   // movePath.pathDataArray[4].commands[17].cmdParameters.pickAndPlaceParameters.targetParameter.direction[1..3] := 0.0;
   // movePath.pathDataArray[4].commands[18].cmdParameters.pickAndPlaceParameters.targetParameter.direction[1..3] := 0.0;
   // movePath.pathDataArray[4].commands[19].cmdParameters.pickAndPlaceParameters.targetParameter.direction[1..3] := 0.0;
   // movePath.pathDataArray[4].commands[20].cmdParameters.pickAndPlaceParameters.targetParameter.direction[1..3] := 0.0;
   // movePath.pathDataArray[5].commands[1].cmdParameters.pickAndPlaceParameters.targetParameter.direction[1..3] := 0.0;
   // movePath.pathDataArray[5].commands[2].cmdParameters.pickAndPlaceParameters.targetParameter.direction[1..3] := 0.0;
   // movePath.pathDataArray[5].commands[3].cmdParameters.pickAndPlaceParameters.targetParameter.direction[1..3] := 0.0;
   // movePath.pathDataArray[5].commands[4].cmdParameters.pickAndPlaceParameters.targetParameter.direction[1..3] := 0.0;
   // movePath.pathDataArray[5].commands[5].cmdParameters.pickAndPlaceParameters.targetParameter.direction[1..3] := 0.0;
   // movePath.pathDataArray[5].commands[6].cmdParameters.pickAndPlaceParameters.targetParameter.direction[1..3] := 0.0;
   // movePath.pathDataArray[5].commands[7].cmdParameters.pickAndPlaceParameters.targetParameter.direction[1..3] := 0.0;
   // movePath.pathDataArray[5].commands[8].cmdParameters.pickAndPlaceParameters.targetParameter.direction[1..3] := 0.0;
   // movePath.pathDataArray[5].commands[9].cmdParameters.pickAndPlaceParameters.targetParameter.direction[1..3] := 0.0;
   // movePath.pathDataArray[5].commands[10].cmdParameters.pickAndPlaceParameters.targetParameter.direction[1..3] := 0.0;
   // movePath.pathDataArray[5].commands[11].cmdParameters.pickAndPlaceParameters.targetParameter.direction[1..3] := 0.0;
   // movePath.pathDataArray[5].commands[12].cmdParameters.pickAndPlaceParameters.targetParameter.direction[1..3] := 0.0;
   // movePath.pathDataArray[5].commands[13].cmdParameters.pickAndPlaceParameters.targetParameter.direction[1..3] := 0.0;
   // movePath.pathDataArray[5].commands[14].cmdParameters.pickAndPlaceParameters.targetParameter.direction[1..3] := 0.0;
   // movePath.pathDataArray[5].commands[15].cmdParameters.pickAndPlaceParameters.targetParameter.direction[1..3] := 0.0;
   // movePath.pathDataArray[5].commands[16].cmdParameters.pickAndPlaceParameters.targetParameter.direction[1..3] := 0.0;
   // movePath.pathDataArray[5].commands[17].cmdParameters.pickAndPlaceParameters.targetParameter.direction[1..3] := 0.0;
   // movePath.pathDataArray[5].commands[18].cmdParameters.pickAndPlaceParameters.targetParameter.direction[1..3] := 0.0;
   // movePath.pathDataArray[5].commands[19].cmdParameters.pickAndPlaceParameters.targetParameter.direction[1..3] := 0.0;
   // movePath.pathDataArray[5].commands[20].cmdParameters.pickAndPlaceParameters.targetParameter.direction[1..3] := 0.0;
   // movePath.pathDataArray[1].commands[1..20].cmdParameters.pickAndPlaceParameters.targetParameter.workingHeight := 0.0;
   // movePath.pathDataArray[2].commands[1..20].cmdParameters.pickAndPlaceParameters.targetParameter.workingHeight := 0.0;
   // movePath.pathDataArray[3].commands[1..20].cmdParameters.pickAndPlaceParameters.targetParameter.workingHeight := 0.0;
   // movePath.pathDataArray[4].commands[1].cmdParameters.pickAndPlaceParameters.targetParameter.workingHeight := 0.0;
   // movePath.pathDataArray[4].commands[2].cmdParameters.pickAndPlaceParameters.targetParameter.workingHeight := 60.0;
   // movePath.pathDataArray[4].commands[3].cmdParameters.pickAndPlaceParameters.targetParameter.workingHeight := 0.0;
   // movePath.pathDataArray[4].commands[4].cmdParameters.pickAndPlaceParameters.targetParameter.workingHeight := 60.0;
   // movePath.pathDataArray[4].commands[5..20].cmdParameters.pickAndPlaceParameters.targetParameter.workingHeight := 0.0;
   // movePath.pathDataArray[5].commands[1..20].cmdParameters.pickAndPlaceParameters.targetParameter.workingHeight := 0.0;
   // movePath.pathDataArray[1].commands[1..20].cmdParameters.pickAndPlaceParameters.targetParameter.transitionArea := 0.0;
   // movePath.pathDataArray[2].commands[1..20].cmdParameters.pickAndPlaceParameters.targetParameter.transitionArea := 0.0;
   // movePath.pathDataArray[3].commands[1..20].cmdParameters.pickAndPlaceParameters.targetParameter.transitionArea := 0.0;
   // movePath.pathDataArray[4].commands[1..20].cmdParameters.pickAndPlaceParameters.targetParameter.transitionArea := 0.0;
   // movePath.pathDataArray[5].commands[1..20].cmdParameters.pickAndPlaceParameters.targetParameter.transitionArea := 0.0;
   // movePath.pathDataArray[1].commands[1..20].cmdParameters.pickAndPlaceParameters.targetParameter.dynamicsFactor := 100.0;
   // movePath.pathDataArray[2].commands[1..20].cmdParameters.pickAndPlaceParameters.targetParameter.dynamicsFactor := 100.0;
   // movePath.pathDataArray[3].commands[1..20].cmdParameters.pickAndPlaceParameters.targetParameter.dynamicsFactor := 100.0;
   // movePath.pathDataArray[4].commands[1..20].cmdParameters.pickAndPlaceParameters.targetParameter.dynamicsFactor := 100.0;
   // movePath.pathDataArray[5].commands[1..20].cmdParameters.pickAndPlaceParameters.targetParameter.dynamicsFactor := 100.0;
   // movePath.pathDataArray[1].commands[1].setFlags[1].flag := 1;
   // movePath.pathDataArray[1].commands[1].setFlags[2..3].flag := -1;
   // movePath.pathDataArray[1].commands[2].setFlags[1..3].flag := -1;
   // movePath.pathDataArray[1].commands[3].setFlags[1].flag := 0;
   // movePath.pathDataArray[1].commands[3].setFlags[2].flag := 1;
   // movePath.pathDataArray[1].commands[3].setFlags[3].flag := -1;
   // movePath.pathDataArray[1].commands[4].setFlags[1..3].flag := -1;
   // movePath.pathDataArray[1].commands[5].setFlags[1..3].flag := -1;
   // movePath.pathDataArray[1].commands[6].setFlags[1..3].flag := -1;
   // movePath.pathDataArray[1].commands[7].setFlags[1].flag := 0;
   // movePath.pathDataArray[1].commands[7].setFlags[2..3].flag := -1;
   // movePath.pathDataArray[1].commands[8].setFlags[1..3].flag := -1;
   // movePath.pathDataArray[1].commands[9].setFlags[1].flag := 1;
   // movePath.pathDataArray[1].commands[9].setFlags[2..3].flag := -1;
   // movePath.pathDataArray[1].commands[10].setFlags[1..3].flag := -1;
   // movePath.pathDataArray[1].commands[11].setFlags[1..3].flag := -1;
   // movePath.pathDataArray[1].commands[12].setFlags[1..3].flag := -1;
   // movePath.pathDataArray[1].commands[13].setFlags[1..3].flag := -1;
   // movePath.pathDataArray[1].commands[14].setFlags[1..3].flag := -1;
   // movePath.pathDataArray[1].commands[15].setFlags[1..3].flag := -1;
   // movePath.pathDataArray[1].commands[16].setFlags[1..3].flag := -1;
   // movePath.pathDataArray[1].commands[17].setFlags[1..3].flag := -1;
   // movePath.pathDataArray[1].commands[18].setFlags[1..3].flag := -1;
   // movePath.pathDataArray[1].commands[19].setFlags[1..3].flag := -1;
   // movePath.pathDataArray[1].commands[20].setFlags[1..3].flag := -1;
   // movePath.pathDataArray[2].commands[1].setFlags[1..3].flag := -1;
   // movePath.pathDataArray[2].commands[2].setFlags[1].flag := 1;
   // movePath.pathDataArray[2].commands[2].setFlags[2..3].flag := -1;
   // movePath.pathDataArray[2].commands[3].setFlags[1..3].flag := -1;
   // movePath.pathDataArray[2].commands[4].setFlags[1].flag := 0;
   // movePath.pathDataArray[2].commands[4].setFlags[2].flag := 1;
   // movePath.pathDataArray[2].commands[4].setFlags[3].flag := -1;
   // movePath.pathDataArray[2].commands[5].setFlags[1..3].flag := -1;
   // movePath.pathDataArray[2].commands[6].setFlags[1..3].flag := -1;
   // movePath.pathDataArray[2].commands[7].setFlags[1..3].flag := -1;
   // movePath.pathDataArray[2].commands[8].setFlags[1].flag := 0;
   // movePath.pathDataArray[2].commands[8].setFlags[2..3].flag := -1;
   // movePath.pathDataArray[2].commands[9].setFlags[1..3].flag := -1;
   // movePath.pathDataArray[2].commands[10].setFlags[1].flag := 1;
   // movePath.pathDataArray[2].commands[10].setFlags[2..3].flag := -1;
   // movePath.pathDataArray[2].commands[11].setFlags[1..3].flag := -1;
   // movePath.pathDataArray[2].commands[12].setFlags[1..3].flag := -1;
   // movePath.pathDataArray[2].commands[13].setFlags[1..3].flag := -1;
   // movePath.pathDataArray[2].commands[14].setFlags[1..3].flag := -1;
   // movePath.pathDataArray[2].commands[15].setFlags[1..3].flag := -1;
   // movePath.pathDataArray[2].commands[16].setFlags[1..3].flag := -1;
   // movePath.pathDataArray[2].commands[17].setFlags[1..3].flag := -1;
   // movePath.pathDataArray[2].commands[18].setFlags[1..3].flag := -1;
   // movePath.pathDataArray[2].commands[19].setFlags[1..3].flag := -1;
   // movePath.pathDataArray[2].commands[20].setFlags[1..3].flag := -1;
   // movePath.pathDataArray[3].commands[1].setFlags[1].flag := 2;
   // movePath.pathDataArray[3].commands[1].setFlags[2].flag := 3;
   // movePath.pathDataArray[3].commands[1].setFlags[3].flag := -1;
   // movePath.pathDataArray[3].commands[2].setFlags[1].flag := 4;
   // movePath.pathDataArray[3].commands[2].setFlags[2..3].flag := -1;
   // movePath.pathDataArray[3].commands[3].setFlags[1..3].flag := -1;
   // movePath.pathDataArray[3].commands[4].setFlags[1..3].flag := -1;
   // movePath.pathDataArray[3].commands[5].setFlags[1].flag := 3;
   // movePath.pathDataArray[3].commands[5].setFlags[2..3].flag := -1;
   // movePath.pathDataArray[3].commands[6].setFlags[1..3].flag := -1;
   // movePath.pathDataArray[3].commands[7].setFlags[1..3].flag := -1;
   // movePath.pathDataArray[3].commands[8].setFlags[1..3].flag := -1;
   // movePath.pathDataArray[3].commands[9].setFlags[1..3].flag := -1;
   // movePath.pathDataArray[3].commands[10].setFlags[1..3].flag := -1;
   // movePath.pathDataArray[3].commands[11].setFlags[1..3].flag := -1;
   // movePath.pathDataArray[3].commands[12].setFlags[1..3].flag := -1;
   // movePath.pathDataArray[3].commands[13].setFlags[1..3].flag := -1;
   // movePath.pathDataArray[3].commands[14].setFlags[1..3].flag := -1;
   // movePath.pathDataArray[3].commands[15].setFlags[1..3].flag := -1;
   // movePath.pathDataArray[3].commands[16].setFlags[1..3].flag := -1;
   // movePath.pathDataArray[3].commands[17].setFlags[1..3].flag := -1;
   // movePath.pathDataArray[3].commands[18].setFlags[1..3].flag := -1;
   // movePath.pathDataArray[3].commands[19].setFlags[1..3].flag := -1;
   // movePath.pathDataArray[3].commands[20].setFlags[1..3].flag := -1;
   // movePath.pathDataArray[4].commands[1].setFlags[1].flag := 5;
   // movePath.pathDataArray[4].commands[1].setFlags[2..3].flag := -1;
   // movePath.pathDataArray[4].commands[2].setFlags[1].flag := -1;
   // movePath.pathDataArray[4].commands[2].setFlags[2].flag := 5;
   // movePath.pathDataArray[4].commands[2].setFlags[3].flag := -1;
   // movePath.pathDataArray[4].commands[3].setFlags[1..3].flag := -1;
   // movePath.pathDataArray[4].commands[4].setFlags[1..3].flag := -1;
   // movePath.pathDataArray[4].commands[5].setFlags[1..3].flag := -1;
   // movePath.pathDataArray[4].commands[6].setFlags[1..3].flag := -1;
   // movePath.pathDataArray[4].commands[7].setFlags[1..3].flag := -1;
   // movePath.pathDataArray[4].commands[8].setFlags[1..3].flag := -1;
   // movePath.pathDataArray[4].commands[9].setFlags[1..3].flag := -1;
   // movePath.pathDataArray[4].commands[10].setFlags[1..3].flag := -1;
   // movePath.pathDataArray[4].commands[11].setFlags[1..3].flag := -1;
   // movePath.pathDataArray[4].commands[12].setFlags[1..3].flag := -1;
   // movePath.pathDataArray[4].commands[13].setFlags[1..3].flag := -1;
   // movePath.pathDataArray[4].commands[14].setFlags[1..3].flag := -1;
   // movePath.pathDataArray[4].commands[15].setFlags[1..3].flag := -1;
   // movePath.pathDataArray[4].commands[16].setFlags[1..3].flag := -1;
   // movePath.pathDataArray[4].commands[17].setFlags[1..3].flag := -1;
   // movePath.pathDataArray[4].commands[18].setFlags[1..3].flag := -1;
   // movePath.pathDataArray[4].commands[19].setFlags[1..3].flag := -1;
   // movePath.pathDataArray[4].commands[20].setFlags[1..3].flag := -1;
   // movePath.pathDataArray[5].commands[1].setFlags[1..3].flag := -1;
   // movePath.pathDataArray[5].commands[2].setFlags[1..3].flag := -1;
   // movePath.pathDataArray[5].commands[3].setFlags[1..3].flag := -1;
   // movePath.pathDataArray[5].commands[4].setFlags[1..3].flag := -1;
   // movePath.pathDataArray[5].commands[5].setFlags[1..3].flag := -1;
   // movePath.pathDataArray[5].commands[6].setFlags[1..3].flag := -1;
   // movePath.pathDataArray[5].commands[7].setFlags[1..3].flag := -1;
   // movePath.pathDataArray[5].commands[8].setFlags[1..3].flag := -1;
   // movePath.pathDataArray[5].commands[9].setFlags[1..3].flag := -1;
   // movePath.pathDataArray[5].commands[10].setFlags[1..3].flag := -1;
   // movePath.pathDataArray[5].commands[11].setFlags[1..3].flag := -1;
   // movePath.pathDataArray[5].commands[12].setFlags[1..3].flag := -1;
   // movePath.pathDataArray[5].commands[13].setFlags[1..3].flag := -1;
   // movePath.pathDataArray[5].commands[14].setFlags[1..3].flag := -1;
   // movePath.pathDataArray[5].commands[15].setFlags[1..3].flag := -1;
   // movePath.pathDataArray[5].commands[16].setFlags[1..3].flag := -1;
   // movePath.pathDataArray[5].commands[17].setFlags[1..3].flag := -1;
   // movePath.pathDataArray[5].commands[18].setFlags[1..3].flag := -1;
   // movePath.pathDataArray[5].commands[19].setFlags[1..3].flag := -1;
   // movePath.pathDataArray[5].commands[20].setFlags[1..3].flag := -1;
   // movePath.pathDataArray[1].commands[1].setFlags[1].flagMode := 1;
   // movePath.pathDataArray[1].commands[1].setFlags[2..3].flagMode := 0;
   // movePath.pathDataArray[1].commands[2].setFlags[1..3].flagMode := 1;
   // movePath.pathDataArray[1].commands[3].setFlags[1].flagMode := 1;
   // movePath.pathDataArray[1].commands[3].setFlags[2].flagMode := 11;
   // movePath.pathDataArray[1].commands[3].setFlags[3].flagMode := 1;
   // movePath.pathDataArray[1].commands[4].setFlags[1..3].flagMode := 1;
   // movePath.pathDataArray[1].commands[5].setFlags[1..3].flagMode := 1;
   // movePath.pathDataArray[1].commands[6].setFlags[1..3].flagMode := 1;
   // movePath.pathDataArray[1].commands[7].setFlags[1].flagMode := 1;
   // movePath.pathDataArray[1].commands[7].setFlags[2..3].flagMode := 0;
   // movePath.pathDataArray[1].commands[8].setFlags[1..3].flagMode := 0;
   // movePath.pathDataArray[1].commands[9].setFlags[1].flagMode := 11;
   // movePath.pathDataArray[1].commands[9].setFlags[2..3].flagMode := 0;
   // movePath.pathDataArray[1].commands[10].setFlags[1..3].flagMode := 1;
   // movePath.pathDataArray[1].commands[11].setFlags[1..3].flagMode := 1;
   // movePath.pathDataArray[1].commands[12].setFlags[1..3].flagMode := 1;
   // movePath.pathDataArray[1].commands[13].setFlags[1..3].flagMode := 1;
   // movePath.pathDataArray[1].commands[14].setFlags[1..3].flagMode := 1;
   // movePath.pathDataArray[1].commands[15].setFlags[1..3].flagMode := 1;
   // movePath.pathDataArray[1].commands[16].setFlags[1..3].flagMode := 1;
   // movePath.pathDataArray[1].commands[17].setFlags[1..3].flagMode := 1;
   // movePath.pathDataArray[1].commands[18].setFlags[1..3].flagMode := 1;
   // movePath.pathDataArray[1].commands[19].setFlags[1..3].flagMode := 1;
   // movePath.pathDataArray[1].commands[20].setFlags[1..3].flagMode := 1;
   // movePath.pathDataArray[2].commands[1].setFlags[1..3].flagMode := 1;
   // movePath.pathDataArray[2].commands[2].setFlags[1].flagMode := 1;
   // movePath.pathDataArray[2].commands[2].setFlags[2..3].flagMode := 0;
   // movePath.pathDataArray[2].commands[3].setFlags[1..3].flagMode := 1;
   // movePath.pathDataArray[2].commands[4].setFlags[1].flagMode := 1;
   // movePath.pathDataArray[2].commands[4].setFlags[2].flagMode := 11;
   // movePath.pathDataArray[2].commands[4].setFlags[3].flagMode := 1;
   // movePath.pathDataArray[2].commands[5].setFlags[1..3].flagMode := 1;
   // movePath.pathDataArray[2].commands[6].setFlags[1..3].flagMode := 1;
   // movePath.pathDataArray[2].commands[7].setFlags[1..3].flagMode := 1;
   // movePath.pathDataArray[2].commands[8].setFlags[1].flagMode := 1;
   // movePath.pathDataArray[2].commands[8].setFlags[2..3].flagMode := 0;
   // movePath.pathDataArray[2].commands[9].setFlags[1..3].flagMode := 0;
   // movePath.pathDataArray[2].commands[10].setFlags[1].flagMode := 11;
   // movePath.pathDataArray[2].commands[10].setFlags[2..3].flagMode := 0;
   // movePath.pathDataArray[2].commands[11].setFlags[1..3].flagMode := 1;
   // movePath.pathDataArray[2].commands[12].setFlags[1..3].flagMode := 1;
   // movePath.pathDataArray[2].commands[13].setFlags[1..3].flagMode := 1;
   // movePath.pathDataArray[2].commands[14].setFlags[1..3].flagMode := 1;
   // movePath.pathDataArray[2].commands[15].setFlags[1..3].flagMode := 1;
   // movePath.pathDataArray[2].commands[16].setFlags[1..3].flagMode := 1;
   // movePath.pathDataArray[2].commands[17].setFlags[1..3].flagMode := 1;
   // movePath.pathDataArray[2].commands[18].setFlags[1..3].flagMode := 1;
   // movePath.pathDataArray[2].commands[19].setFlags[1..3].flagMode := 1;
   // movePath.pathDataArray[2].commands[20].setFlags[1..3].flagMode := 1;
   // movePath.pathDataArray[3].commands[1].setFlags[1].flagMode := 26;
   // movePath.pathDataArray[3].commands[1].setFlags[2..3].flagMode := 1;
   // movePath.pathDataArray[3].commands[2].setFlags[1].flagMode := 11;
   // movePath.pathDataArray[3].commands[2].setFlags[2..3].flagMode := 1;
   // movePath.pathDataArray[3].commands[3].setFlags[1..3].flagMode := 1;
   // movePath.pathDataArray[3].commands[4].setFlags[1..3].flagMode := 1;
   // movePath.pathDataArray[3].commands[5].setFlags[1].flagMode := 11;
   // movePath.pathDataArray[3].commands[5].setFlags[2..3].flagMode := 1;
   // movePath.pathDataArray[3].commands[6].setFlags[1..3].flagMode := 1;
   // movePath.pathDataArray[3].commands[7].setFlags[1..3].flagMode := 1;
   // movePath.pathDataArray[3].commands[8].setFlags[1..3].flagMode := 1;
   // movePath.pathDataArray[3].commands[9].setFlags[1..3].flagMode := 1;
   // movePath.pathDataArray[3].commands[10].setFlags[1..3].flagMode := 1;
   // movePath.pathDataArray[3].commands[11].setFlags[1..3].flagMode := 1;
   // movePath.pathDataArray[3].commands[12].setFlags[1..3].flagMode := 1;
   // movePath.pathDataArray[3].commands[13].setFlags[1..3].flagMode := 1;
   // movePath.pathDataArray[3].commands[14].setFlags[1..3].flagMode := 1;
   // movePath.pathDataArray[3].commands[15].setFlags[1..3].flagMode := 1;
   // movePath.pathDataArray[3].commands[16].setFlags[1..3].flagMode := 1;
   // movePath.pathDataArray[3].commands[17].setFlags[1..3].flagMode := 1;
   // movePath.pathDataArray[3].commands[18].setFlags[1..3].flagMode := 1;
   // movePath.pathDataArray[3].commands[19].setFlags[1..3].flagMode := 1;
   // movePath.pathDataArray[3].commands[20].setFlags[1..3].flagMode := 1;
   // movePath.pathDataArray[4].commands[1].setFlags[1].flagMode := 26;
   // movePath.pathDataArray[4].commands[1].setFlags[2..3].flagMode := 1;
   // movePath.pathDataArray[4].commands[2].setFlags[1].flagMode := 1;
   // movePath.pathDataArray[4].commands[2].setFlags[2].flagMode := 21;
   // movePath.pathDataArray[4].commands[2].setFlags[3].flagMode := 1;
   // movePath.pathDataArray[4].commands[3].setFlags[1..3].flagMode := 1;
   // movePath.pathDataArray[4].commands[4].setFlags[1..3].flagMode := 1;
   // movePath.pathDataArray[4].commands[5].setFlags[1..3].flagMode := 1;
   // movePath.pathDataArray[4].commands[6].setFlags[1..3].flagMode := 1;
   // movePath.pathDataArray[4].commands[7].setFlags[1..3].flagMode := 1;
   // movePath.pathDataArray[4].commands[8].setFlags[1..3].flagMode := 1;
   // movePath.pathDataArray[4].commands[9].setFlags[1..3].flagMode := 1;
   // movePath.pathDataArray[4].commands[10].setFlags[1..3].flagMode := 1;
   // movePath.pathDataArray[4].commands[11].setFlags[1..3].flagMode := 1;
   // movePath.pathDataArray[4].commands[12].setFlags[1..3].flagMode := 1;
   // movePath.pathDataArray[4].commands[13].setFlags[1..3].flagMode := 1;
   // movePath.pathDataArray[4].commands[14].setFlags[1..3].flagMode := 1;
   // movePath.pathDataArray[4].commands[15].setFlags[1..3].flagMode := 1;
   // movePath.pathDataArray[4].commands[16].setFlags[1..3].flagMode := 1;
   // movePath.pathDataArray[4].commands[17].setFlags[1..3].flagMode := 1;
   // movePath.pathDataArray[4].commands[18].setFlags[1..3].flagMode := 1;
   // movePath.pathDataArray[4].commands[19].setFlags[1..3].flagMode := 1;
   // movePath.pathDataArray[4].commands[20].setFlags[1..3].flagMode := 1;
   // movePath.pathDataArray[5].commands[1].setFlags[1..3].flagMode := 1;
   // movePath.pathDataArray[5].commands[2].setFlags[1..3].flagMode := 1;
   // movePath.pathDataArray[5].commands[3].setFlags[1..3].flagMode := 1;
   // movePath.pathDataArray[5].commands[4].setFlags[1..3].flagMode := 1;
   // movePath.pathDataArray[5].commands[5].setFlags[1..3].flagMode := 1;
   // movePath.pathDataArray[5].commands[6].setFlags[1..3].flagMode := 1;
   // movePath.pathDataArray[5].commands[7].setFlags[1..3].flagMode := 1;
   // movePath.pathDataArray[5].commands[8].setFlags[1..3].flagMode := 1;
   // movePath.pathDataArray[5].commands[9].setFlags[1..3].flagMode := 1;
   // movePath.pathDataArray[5].commands[10].setFlags[1..3].flagMode := 1;
   // movePath.pathDataArray[5].commands[11].setFlags[1..3].flagMode := 1;
   // movePath.pathDataArray[5].commands[12].setFlags[1..3].flagMode := 1;
   // movePath.pathDataArray[5].commands[13].setFlags[1..3].flagMode := 1;
   // movePath.pathDataArray[5].commands[14].setFlags[1..3].flagMode := 1;
   // movePath.pathDataArray[5].commands[15].setFlags[1..3].flagMode := 1;
   // movePath.pathDataArray[5].commands[16].setFlags[1..3].flagMode := 1;
   // movePath.pathDataArray[5].commands[17].setFlags[1..3].flagMode := 1;
   // movePath.pathDataArray[5].commands[18].setFlags[1..3].flagMode := 1;
   // movePath.pathDataArray[5].commands[19].setFlags[1..3].flagMode := 1;
   // movePath.pathDataArray[5].commands[20].setFlags[1..3].flagMode := 1;
   // movePath.pathDataArray[1].commands[1].setFlags[1..3].remainingDistance := -1.0;
   // movePath.pathDataArray[1].commands[2].setFlags[1..3].remainingDistance := -1.0;
   // movePath.pathDataArray[1].commands[3].setFlags[1..3].remainingDistance := -1.0;
   // movePath.pathDataArray[1].commands[4].setFlags[1..3].remainingDistance := -1.0;
   // movePath.pathDataArray[1].commands[5].setFlags[1..3].remainingDistance := -1.0;
   // movePath.pathDataArray[1].commands[6].setFlags[1..3].remainingDistance := -1.0;
   // movePath.pathDataArray[1].commands[7].setFlags[1..3].remainingDistance := -1.0;
   // movePath.pathDataArray[1].commands[8].setFlags[1..3].remainingDistance := -1.0;
   // movePath.pathDataArray[1].commands[9].setFlags[1..3].remainingDistance := -1.0;
   // movePath.pathDataArray[1].commands[10].setFlags[1..3].remainingDistance := 0.0;
   // movePath.pathDataArray[1].commands[11].setFlags[1..3].remainingDistance := -1.0;
   // movePath.pathDataArray[1].commands[12].setFlags[1..3].remainingDistance := -1.0;
   // movePath.pathDataArray[1].commands[13].setFlags[1..3].remainingDistance := -1.0;
   // movePath.pathDataArray[1].commands[14].setFlags[1..3].remainingDistance := -1.0;
   // movePath.pathDataArray[1].commands[15].setFlags[1..3].remainingDistance := -1.0;
   // movePath.pathDataArray[1].commands[16].setFlags[1..3].remainingDistance := -1.0;
   // movePath.pathDataArray[1].commands[17].setFlags[1..3].remainingDistance := -1.0;
   // movePath.pathDataArray[1].commands[18].setFlags[1..3].remainingDistance := -1.0;
   // movePath.pathDataArray[1].commands[19].setFlags[1..3].remainingDistance := -1.0;
   // movePath.pathDataArray[1].commands[20].setFlags[1..3].remainingDistance := -1.0;
   // movePath.pathDataArray[2].commands[1].setFlags[1..3].remainingDistance := -1.0;
   // movePath.pathDataArray[2].commands[2].setFlags[1..3].remainingDistance := -1.0;
   // movePath.pathDataArray[2].commands[3].setFlags[1..3].remainingDistance := -1.0;
   // movePath.pathDataArray[2].commands[4].setFlags[1..3].remainingDistance := -1.0;
   // movePath.pathDataArray[2].commands[5].setFlags[1..3].remainingDistance := -1.0;
   // movePath.pathDataArray[2].commands[6].setFlags[1..3].remainingDistance := -1.0;
   // movePath.pathDataArray[2].commands[7].setFlags[1..3].remainingDistance := -1.0;
   // movePath.pathDataArray[2].commands[8].setFlags[1..3].remainingDistance := -1.0;
   // movePath.pathDataArray[2].commands[9].setFlags[1..3].remainingDistance := -1.0;
   // movePath.pathDataArray[2].commands[10].setFlags[1..3].remainingDistance := -1.0;
   // movePath.pathDataArray[2].commands[11].setFlags[1..3].remainingDistance := 0.0;
   // movePath.pathDataArray[2].commands[12].setFlags[1..3].remainingDistance := -1.0;
   // movePath.pathDataArray[2].commands[13].setFlags[1..3].remainingDistance := -1.0;
   // movePath.pathDataArray[2].commands[14].setFlags[1..3].remainingDistance := -1.0;
   // movePath.pathDataArray[2].commands[15].setFlags[1..3].remainingDistance := -1.0;
   // movePath.pathDataArray[2].commands[16].setFlags[1..3].remainingDistance := -1.0;
   // movePath.pathDataArray[2].commands[17].setFlags[1..3].remainingDistance := -1.0;
   // movePath.pathDataArray[2].commands[18].setFlags[1..3].remainingDistance := -1.0;
   // movePath.pathDataArray[2].commands[19].setFlags[1..3].remainingDistance := -1.0;
   // movePath.pathDataArray[2].commands[20].setFlags[1..3].remainingDistance := -1.0;
   // movePath.pathDataArray[3].commands[1].setFlags[1..3].remainingDistance := -1.0;
   // movePath.pathDataArray[3].commands[2].setFlags[1..3].remainingDistance := -1.0;
   // movePath.pathDataArray[3].commands[3].setFlags[1..3].remainingDistance := -1.0;
   // movePath.pathDataArray[3].commands[4].setFlags[1..3].remainingDistance := -1.0;
   // movePath.pathDataArray[3].commands[5].setFlags[1..3].remainingDistance := -1.0;
   // movePath.pathDataArray[3].commands[6].setFlags[1..3].remainingDistance := -1.0;
   // movePath.pathDataArray[3].commands[7].setFlags[1..3].remainingDistance := -1.0;
   // movePath.pathDataArray[3].commands[8].setFlags[1..3].remainingDistance := -1.0;
   // movePath.pathDataArray[3].commands[9].setFlags[1..3].remainingDistance := -1.0;
   // movePath.pathDataArray[3].commands[10].setFlags[1..3].remainingDistance := -1.0;
   // movePath.pathDataArray[3].commands[11].setFlags[1..3].remainingDistance := -1.0;
   // movePath.pathDataArray[3].commands[12].setFlags[1..3].remainingDistance := -1.0;
   // movePath.pathDataArray[3].commands[13].setFlags[1..3].remainingDistance := -1.0;
   // movePath.pathDataArray[3].commands[14].setFlags[1..3].remainingDistance := -1.0;
   // movePath.pathDataArray[3].commands[15].setFlags[1..3].remainingDistance := -1.0;
   // movePath.pathDataArray[3].commands[16].setFlags[1..3].remainingDistance := -1.0;
   // movePath.pathDataArray[3].commands[17].setFlags[1..3].remainingDistance := -1.0;
   // movePath.pathDataArray[3].commands[18].setFlags[1..3].remainingDistance := -1.0;
   // movePath.pathDataArray[3].commands[19].setFlags[1..3].remainingDistance := -1.0;
   // movePath.pathDataArray[3].commands[20].setFlags[1..3].remainingDistance := -1.0;
   // movePath.pathDataArray[4].commands[1].setFlags[1..3].remainingDistance := -1.0;
   // movePath.pathDataArray[4].commands[2].setFlags[1..3].remainingDistance := -1.0;
   // movePath.pathDataArray[4].commands[3].setFlags[1..3].remainingDistance := -1.0;
   // movePath.pathDataArray[4].commands[4].setFlags[1..3].remainingDistance := -1.0;
   // movePath.pathDataArray[4].commands[5].setFlags[1..3].remainingDistance := -1.0;
   // movePath.pathDataArray[4].commands[6].setFlags[1..3].remainingDistance := -1.0;
   // movePath.pathDataArray[4].commands[7].setFlags[1..3].remainingDistance := -1.0;
   // movePath.pathDataArray[4].commands[8].setFlags[1..3].remainingDistance := -1.0;
   // movePath.pathDataArray[4].commands[9].setFlags[1..3].remainingDistance := -1.0;
   // movePath.pathDataArray[4].commands[10].setFlags[1..3].remainingDistance := -1.0;
   // movePath.pathDataArray[4].commands[11].setFlags[1..3].remainingDistance := -1.0;
   // movePath.pathDataArray[4].commands[12].setFlags[1..3].remainingDistance := -1.0;
   // movePath.pathDataArray[4].commands[13].setFlags[1..3].remainingDistance := -1.0;
   // movePath.pathDataArray[4].commands[14].setFlags[1..3].remainingDistance := -1.0;
   // movePath.pathDataArray[4].commands[15].setFlags[1..3].remainingDistance := -1.0;
   // movePath.pathDataArray[4].commands[16].setFlags[1..3].remainingDistance := -1.0;
   // movePath.pathDataArray[4].commands[17].setFlags[1..3].remainingDistance := -1.0;
   // movePath.pathDataArray[4].commands[18].setFlags[1..3].remainingDistance := -1.0;
   // movePath.pathDataArray[4].commands[19].setFlags[1..3].remainingDistance := -1.0;
   // movePath.pathDataArray[4].commands[20].setFlags[1..3].remainingDistance := -1.0;
   // movePath.pathDataArray[5].commands[1].setFlags[1..3].remainingDistance := -1.0;
   // movePath.pathDataArray[5].commands[2].setFlags[1..3].remainingDistance := -1.0;
   // movePath.pathDataArray[5].commands[3].setFlags[1..3].remainingDistance := -1.0;
   // movePath.pathDataArray[5].commands[4].setFlags[1..3].remainingDistance := -1.0;
   // movePath.pathDataArray[5].commands[5].setFlags[1..3].remainingDistance := -1.0;
   // movePath.pathDataArray[5].commands[6].setFlags[1..3].remainingDistance := -1.0;
   // movePath.pathDataArray[5].commands[7].setFlags[1..3].remainingDistance := -1.0;
   // movePath.pathDataArray[5].commands[8].setFlags[1..3].remainingDistance := -1.0;
   // movePath.pathDataArray[5].commands[9].setFlags[1..3].remainingDistance := -1.0;
   // movePath.pathDataArray[5].commands[10].setFlags[1..3].remainingDistance := -1.0;
   // movePath.pathDataArray[5].commands[11].setFlags[1..3].remainingDistance := -1.0;
   // movePath.pathDataArray[5].commands[12].setFlags[1..3].remainingDistance := -1.0;
   // movePath.pathDataArray[5].commands[13].setFlags[1..3].remainingDistance := -1.0;
   // movePath.pathDataArray[5].commands[14].setFlags[1..3].remainingDistance := -1.0;
   // movePath.pathDataArray[5].commands[15].setFlags[1..3].remainingDistance := -1.0;
   // movePath.pathDataArray[5].commands[16].setFlags[1..3].remainingDistance := -1.0;
   // movePath.pathDataArray[5].commands[17].setFlags[1..3].remainingDistance := -1.0;
   // movePath.pathDataArray[5].commands[18].setFlags[1..3].remainingDistance := -1.0;
   // movePath.pathDataArray[5].commands[19].setFlags[1..3].remainingDistance := -1.0;
   // movePath.pathDataArray[5].commands[20].setFlags[1..3].remainingDistance := -1.0;
   // movePath.pathDataArray[1].commands[1].valueFlags[1..4].flag := -1;
   // movePath.pathDataArray[1].commands[2].valueFlags[1..4].flag := -1;
   // movePath.pathDataArray[1].commands[3].valueFlags[1..4].flag := -1;
   // movePath.pathDataArray[1].commands[4].valueFlags[1..4].flag := -1;
   // movePath.pathDataArray[1].commands[5].valueFlags[1..4].flag := -1;
   // movePath.pathDataArray[1].commands[6].valueFlags[1..4].flag := -1;
   // movePath.pathDataArray[1].commands[7].valueFlags[1..4].flag := -1;
   // movePath.pathDataArray[1].commands[8].valueFlags[1..4].flag := -1;
   // movePath.pathDataArray[1].commands[9].valueFlags[1..4].flag := -1;
   // movePath.pathDataArray[1].commands[10].valueFlags[1..4].flag := -1;
   // movePath.pathDataArray[1].commands[11].valueFlags[1..4].flag := -1;
   // movePath.pathDataArray[1].commands[12].valueFlags[1..4].flag := -1;
   // movePath.pathDataArray[1].commands[13].valueFlags[1..4].flag := -1;
   // movePath.pathDataArray[1].commands[14].valueFlags[1..4].flag := -1;
   // movePath.pathDataArray[1].commands[15].valueFlags[1..4].flag := -1;
   // movePath.pathDataArray[1].commands[16].valueFlags[1..4].flag := -1;
   // movePath.pathDataArray[1].commands[17].valueFlags[1..4].flag := -1;
   // movePath.pathDataArray[1].commands[18].valueFlags[1..4].flag := -1;
   // movePath.pathDataArray[1].commands[19].valueFlags[1..4].flag := -1;
   // movePath.pathDataArray[1].commands[20].valueFlags[1..4].flag := -1;
   // movePath.pathDataArray[2].commands[1].valueFlags[1..4].flag := -1;
   // movePath.pathDataArray[2].commands[2].valueFlags[1..4].flag := -1;
   // movePath.pathDataArray[2].commands[3].valueFlags[1..4].flag := -1;
   // movePath.pathDataArray[2].commands[4].valueFlags[1..4].flag := -1;
   // movePath.pathDataArray[2].commands[5].valueFlags[1..4].flag := -1;
   // movePath.pathDataArray[2].commands[6].valueFlags[1..4].flag := -1;
   // movePath.pathDataArray[2].commands[7].valueFlags[1..4].flag := -1;
   // movePath.pathDataArray[2].commands[8].valueFlags[1..4].flag := -1;
   // movePath.pathDataArray[2].commands[9].valueFlags[1..4].flag := -1;
   // movePath.pathDataArray[2].commands[10].valueFlags[1..4].flag := -1;
   // movePath.pathDataArray[2].commands[11].valueFlags[1..4].flag := -1;
   // movePath.pathDataArray[2].commands[12].valueFlags[1..4].flag := -1;
   // movePath.pathDataArray[2].commands[13].valueFlags[1..4].flag := -1;
   // movePath.pathDataArray[2].commands[14].valueFlags[1..4].flag := -1;
   // movePath.pathDataArray[2].commands[15].valueFlags[1..4].flag := -1;
   // movePath.pathDataArray[2].commands[16].valueFlags[1..4].flag := -1;
   // movePath.pathDataArray[2].commands[17].valueFlags[1..4].flag := -1;
   // movePath.pathDataArray[2].commands[18].valueFlags[1..4].flag := -1;
   // movePath.pathDataArray[2].commands[19].valueFlags[1..4].flag := -1;
   // movePath.pathDataArray[2].commands[20].valueFlags[1..4].flag := -1;
   // movePath.pathDataArray[3].commands[1].valueFlags[1..4].flag := -1;
   // movePath.pathDataArray[3].commands[2].valueFlags[1..4].flag := -1;
   // movePath.pathDataArray[3].commands[3].valueFlags[1..4].flag := -1;
   // movePath.pathDataArray[3].commands[4].valueFlags[1..4].flag := -1;
   // movePath.pathDataArray[3].commands[5].valueFlags[1..4].flag := -1;
   // movePath.pathDataArray[3].commands[6].valueFlags[1..4].flag := -1;
   // movePath.pathDataArray[3].commands[7].valueFlags[1..4].flag := -1;
   // movePath.pathDataArray[3].commands[8].valueFlags[1..4].flag := -1;
   // movePath.pathDataArray[3].commands[9].valueFlags[1..4].flag := -1;
   // movePath.pathDataArray[3].commands[10].valueFlags[1..4].flag := -1;
   // movePath.pathDataArray[3].commands[11].valueFlags[1..4].flag := -1;
   // movePath.pathDataArray[3].commands[12].valueFlags[1..4].flag := -1;
   // movePath.pathDataArray[3].commands[13].valueFlags[1..4].flag := -1;
   // movePath.pathDataArray[3].commands[14].valueFlags[1..4].flag := -1;
   // movePath.pathDataArray[3].commands[15].valueFlags[1..4].flag := -1;
   // movePath.pathDataArray[3].commands[16].valueFlags[1..4].flag := -1;
   // movePath.pathDataArray[3].commands[17].valueFlags[1..4].flag := -1;
   // movePath.pathDataArray[3].commands[18].valueFlags[1..4].flag := -1;
   // movePath.pathDataArray[3].commands[19].valueFlags[1..4].flag := -1;
   // movePath.pathDataArray[3].commands[20].valueFlags[1..4].flag := -1;
   // movePath.pathDataArray[4].commands[1].valueFlags[1..4].flag := -1;
   // movePath.pathDataArray[4].commands[2].valueFlags[1..4].flag := -1;
   // movePath.pathDataArray[4].commands[3].valueFlags[1..4].flag := -1;
   // movePath.pathDataArray[4].commands[4].valueFlags[1..4].flag := -1;
   // movePath.pathDataArray[4].commands[5].valueFlags[1..4].flag := -1;
   // movePath.pathDataArray[4].commands[6].valueFlags[1..4].flag := -1;
   // movePath.pathDataArray[4].commands[7].valueFlags[1..4].flag := -1;
   // movePath.pathDataArray[4].commands[8].valueFlags[1..4].flag := -1;
   // movePath.pathDataArray[4].commands[9].valueFlags[1..4].flag := -1;
   // movePath.pathDataArray[4].commands[10].valueFlags[1..4].flag := -1;
   // movePath.pathDataArray[4].commands[11].valueFlags[1..4].flag := -1;
   // movePath.pathDataArray[4].commands[12].valueFlags[1..4].flag := -1;
   // movePath.pathDataArray[4].commands[13].valueFlags[1..4].flag := -1;
   // movePath.pathDataArray[4].commands[14].valueFlags[1..4].flag := -1;
   // movePath.pathDataArray[4].commands[15].valueFlags[1..4].flag := -1;
   // movePath.pathDataArray[4].commands[16].valueFlags[1..4].flag := -1;
   // movePath.pathDataArray[4].commands[17].valueFlags[1..4].flag := -1;
   // movePath.pathDataArray[4].commands[18].valueFlags[1..4].flag := -1;
   // movePath.pathDataArray[4].commands[19].valueFlags[1..4].flag := -1;
   // movePath.pathDataArray[4].commands[20].valueFlags[1..4].flag := -1;
   // movePath.pathDataArray[5].commands[1].valueFlags[1..4].flag := -1;
   // movePath.pathDataArray[5].commands[2].valueFlags[1..4].flag := -1;
   // movePath.pathDataArray[5].commands[3].valueFlags[1..4].flag := -1;
   // movePath.pathDataArray[5].commands[4].valueFlags[1..4].flag := -1;
   // movePath.pathDataArray[5].commands[5].valueFlags[1..4].flag := -1;
   // movePath.pathDataArray[5].commands[6].valueFlags[1..4].flag := -1;
   // movePath.pathDataArray[5].commands[7].valueFlags[1..4].flag := -1;
   // movePath.pathDataArray[5].commands[8].valueFlags[1..4].flag := -1;
   // movePath.pathDataArray[5].commands[9].valueFlags[1..4].flag := -1;
   // movePath.pathDataArray[5].commands[10].valueFlags[1..4].flag := -1;
   // movePath.pathDataArray[5].commands[11].valueFlags[1..4].flag := -1;
   // movePath.pathDataArray[5].commands[12].valueFlags[1..4].flag := -1;
   // movePath.pathDataArray[5].commands[13].valueFlags[1..4].flag := -1;
   // movePath.pathDataArray[5].commands[14].valueFlags[1..4].flag := -1;
   // movePath.pathDataArray[5].commands[15].valueFlags[1..4].flag := -1;
   // movePath.pathDataArray[5].commands[16].valueFlags[1..4].flag := -1;
   // movePath.pathDataArray[5].commands[17].valueFlags[1..4].flag := -1;
   // movePath.pathDataArray[5].commands[18].valueFlags[1..4].flag := -1;
   // movePath.pathDataArray[5].commands[19].valueFlags[1..4].flag := -1;
   // movePath.pathDataArray[5].commands[20].valueFlags[1..4].flag := -1;
   // movePath.pathDataArray[1].commands[1].valueFlags[1..4].value := 0.0;
   // movePath.pathDataArray[1].commands[2].valueFlags[1..4].value := 0.0;
   // movePath.pathDataArray[1].commands[3].valueFlags[1..4].value := 0.0;
   // movePath.pathDataArray[1].commands[4].valueFlags[1..4].value := 0.0;
   // movePath.pathDataArray[1].commands[5].valueFlags[1..4].value := 0.0;
   // movePath.pathDataArray[1].commands[6].valueFlags[1..4].value := 0.0;
   // movePath.pathDataArray[1].commands[7].valueFlags[1..4].value := 0.0;
   // movePath.pathDataArray[1].commands[8].valueFlags[1..4].value := 0.0;
   // movePath.pathDataArray[1].commands[9].valueFlags[1..4].value := 0.0;
   // movePath.pathDataArray[1].commands[10].valueFlags[1..4].value := 0.0;
   // movePath.pathDataArray[1].commands[11].valueFlags[1..4].value := 0.0;
   // movePath.pathDataArray[1].commands[12].valueFlags[1..4].value := 0.0;
   // movePath.pathDataArray[1].commands[13].valueFlags[1..4].value := 0.0;
   // movePath.pathDataArray[1].commands[14].valueFlags[1..4].value := 0.0;
   // movePath.pathDataArray[1].commands[15].valueFlags[1..4].value := 0.0;
   // movePath.pathDataArray[1].commands[16].valueFlags[1..4].value := 0.0;
   // movePath.pathDataArray[1].commands[17].valueFlags[1..4].value := 0.0;
   // movePath.pathDataArray[1].commands[18].valueFlags[1..4].value := 0.0;
   // movePath.pathDataArray[1].commands[19].valueFlags[1..4].value := 0.0;
   // movePath.pathDataArray[1].commands[20].valueFlags[1..4].value := 0.0;
   // movePath.pathDataArray[2].commands[1].valueFlags[1..4].value := 0.0;
   // movePath.pathDataArray[2].commands[2].valueFlags[1..4].value := 0.0;
   // movePath.pathDataArray[2].commands[3].valueFlags[1..4].value := 0.0;
   // movePath.pathDataArray[2].commands[4].valueFlags[1..4].value := 0.0;
   // movePath.pathDataArray[2].commands[5].valueFlags[1..4].value := 0.0;
   // movePath.pathDataArray[2].commands[6].valueFlags[1..4].value := 0.0;
   // movePath.pathDataArray[2].commands[7].valueFlags[1..4].value := 0.0;
   // movePath.pathDataArray[2].commands[8].valueFlags[1..4].value := 0.0;
   // movePath.pathDataArray[2].commands[9].valueFlags[1..4].value := 0.0;
   // movePath.pathDataArray[2].commands[10].valueFlags[1..4].value := 0.0;
   // movePath.pathDataArray[2].commands[11].valueFlags[1..4].value := 0.0;
   // movePath.pathDataArray[2].commands[12].valueFlags[1..4].value := 0.0;
   // movePath.pathDataArray[2].commands[13].valueFlags[1..4].value := 0.0;
   // movePath.pathDataArray[2].commands[14].valueFlags[1..4].value := 0.0;
   // movePath.pathDataArray[2].commands[15].valueFlags[1..4].value := 0.0;
   // movePath.pathDataArray[2].commands[16].valueFlags[1..4].value := 0.0;
   // movePath.pathDataArray[2].commands[17].valueFlags[1..4].value := 0.0;
   // movePath.pathDataArray[2].commands[18].valueFlags[1..4].value := 0.0;
   // movePath.pathDataArray[2].commands[19].valueFlags[1..4].value := 0.0;
   // movePath.pathDataArray[2].commands[20].valueFlags[1..4].value := 0.0;
   // movePath.pathDataArray[3].commands[1].valueFlags[1..4].value := 0.0;
   // movePath.pathDataArray[3].commands[2].valueFlags[1..4].value := 0.0;
   // movePath.pathDataArray[3].commands[3].valueFlags[1..4].value := 0.0;
   // movePath.pathDataArray[3].commands[4].valueFlags[1..4].value := 0.0;
   // movePath.pathDataArray[3].commands[5].valueFlags[1..4].value := 0.0;
   // movePath.pathDataArray[3].commands[6].valueFlags[1..4].value := 0.0;
   // movePath.pathDataArray[3].commands[7].valueFlags[1..4].value := 0.0;
   // movePath.pathDataArray[3].commands[8].valueFlags[1..4].value := 0.0;
   // movePath.pathDataArray[3].commands[9].valueFlags[1..4].value := 0.0;
   // movePath.pathDataArray[3].commands[10].valueFlags[1..4].value := 0.0;
   // movePath.pathDataArray[3].commands[11].valueFlags[1..4].value := 0.0;
   // movePath.pathDataArray[3].commands[12].valueFlags[1..4].value := 0.0;
   // movePath.pathDataArray[3].commands[13].valueFlags[1..4].value := 0.0;
   // movePath.pathDataArray[3].commands[14].valueFlags[1..4].value := 0.0;
   // movePath.pathDataArray[3].commands[15].valueFlags[1..4].value := 0.0;
   // movePath.pathDataArray[3].commands[16].valueFlags[1..4].value := 0.0;
   // movePath.pathDataArray[3].commands[17].valueFlags[1..4].value := 0.0;
   // movePath.pathDataArray[3].commands[18].valueFlags[1..4].value := 0.0;
   // movePath.pathDataArray[3].commands[19].valueFlags[1..4].value := 0.0;
   // movePath.pathDataArray[3].commands[20].valueFlags[1..4].value := 0.0;
   // movePath.pathDataArray[4].commands[1].valueFlags[1..4].value := 0.0;
   // movePath.pathDataArray[4].commands[2].valueFlags[1..4].value := 0.0;
   // movePath.pathDataArray[4].commands[3].valueFlags[1..4].value := 0.0;
   // movePath.pathDataArray[4].commands[4].valueFlags[1..4].value := 0.0;
   // movePath.pathDataArray[4].commands[5].valueFlags[1..4].value := 0.0;
   // movePath.pathDataArray[4].commands[6].valueFlags[1..4].value := 0.0;
   // movePath.pathDataArray[4].commands[7].valueFlags[1..4].value := 0.0;
   // movePath.pathDataArray[4].commands[8].valueFlags[1..4].value := 0.0;
   // movePath.pathDataArray[4].commands[9].valueFlags[1..4].value := 0.0;
   // movePath.pathDataArray[4].commands[10].valueFlags[1..4].value := 0.0;
   // movePath.pathDataArray[4].commands[11].valueFlags[1..4].value := 0.0;
   // movePath.pathDataArray[4].commands[12].valueFlags[1..4].value := 0.0;
   // movePath.pathDataArray[4].commands[13].valueFlags[1..4].value := 0.0;
   // movePath.pathDataArray[4].commands[14].valueFlags[1..4].value := 0.0;
   // movePath.pathDataArray[4].commands[15].valueFlags[1..4].value := 0.0;
   // movePath.pathDataArray[4].commands[16].valueFlags[1..4].value := 0.0;
   // movePath.pathDataArray[4].commands[17].valueFlags[1..4].value := 0.0;
   // movePath.pathDataArray[4].commands[18].valueFlags[1..4].value := 0.0;
   // movePath.pathDataArray[4].commands[19].valueFlags[1..4].value := 0.0;
   // movePath.pathDataArray[4].commands[20].valueFlags[1..4].value := 0.0;
   // movePath.pathDataArray[5].commands[1].valueFlags[1..4].value := 0.0;
   // movePath.pathDataArray[5].commands[2].valueFlags[1..4].value := 0.0;
   // movePath.pathDataArray[5].commands[3].valueFlags[1..4].value := 0.0;
   // movePath.pathDataArray[5].commands[4].valueFlags[1..4].value := 0.0;
   // movePath.pathDataArray[5].commands[5].valueFlags[1..4].value := 0.0;
   // movePath.pathDataArray[5].commands[6].valueFlags[1..4].value := 0.0;
   // movePath.pathDataArray[5].commands[7].valueFlags[1..4].value := 0.0;
   // movePath.pathDataArray[5].commands[8].valueFlags[1..4].value := 0.0;
   // movePath.pathDataArray[5].commands[9].valueFlags[1..4].value := 0.0;
   // movePath.pathDataArray[5].commands[10].valueFlags[1..4].value := 0.0;
   // movePath.pathDataArray[5].commands[11].valueFlags[1..4].value := 0.0;
   // movePath.pathDataArray[5].commands[12].valueFlags[1..4].value := 0.0;
   // movePath.pathDataArray[5].commands[13].valueFlags[1..4].value := 0.0;
   // movePath.pathDataArray[5].commands[14].valueFlags[1..4].value := 0.0;
   // movePath.pathDataArray[5].commands[15].valueFlags[1..4].value := 0.0;
   // movePath.pathDataArray[5].commands[16].valueFlags[1..4].value := 0.0;
   // movePath.pathDataArray[5].commands[17].valueFlags[1..4].value := 0.0;
   // movePath.pathDataArray[5].commands[18].valueFlags[1..4].value := 0.0;
   // movePath.pathDataArray[5].commands[19].valueFlags[1..4].value := 0.0;
   // movePath.pathDataArray[5].commands[20].valueFlags[1..4].value := 0.0;
   // movePath.pathDataArray[1].commands[1].valueFlags[1..4].flagMode := 1;
   // movePath.pathDataArray[1].commands[2].valueFlags[1..4].flagMode := 1;
   // movePath.pathDataArray[1].commands[3].valueFlags[1..4].flagMode := 1;
   // movePath.pathDataArray[1].commands[4].valueFlags[1..4].flagMode := 1;
   // movePath.pathDataArray[1].commands[5].valueFlags[1..4].flagMode := 1;
   // movePath.pathDataArray[1].commands[6].valueFlags[1..4].flagMode := 1;
   // movePath.pathDataArray[1].commands[7].valueFlags[1..4].flagMode := 1;
   // movePath.pathDataArray[1].commands[8].valueFlags[1..4].flagMode := 1;
   // movePath.pathDataArray[1].commands[9].valueFlags[1..4].flagMode := 1;
   // movePath.pathDataArray[1].commands[10].valueFlags[1..4].flagMode := 1;
   // movePath.pathDataArray[1].commands[11].valueFlags[1..4].flagMode := 1;
   // movePath.pathDataArray[1].commands[12].valueFlags[1..4].flagMode := 1;
   // movePath.pathDataArray[1].commands[13].valueFlags[1..4].flagMode := 1;
   // movePath.pathDataArray[1].commands[14].valueFlags[1..4].flagMode := 1;
   // movePath.pathDataArray[1].commands[15].valueFlags[1..4].flagMode := 1;
   // movePath.pathDataArray[1].commands[16].valueFlags[1..4].flagMode := 1;
   // movePath.pathDataArray[1].commands[17].valueFlags[1..4].flagMode := 1;
   // movePath.pathDataArray[1].commands[18].valueFlags[1..4].flagMode := 1;
   // movePath.pathDataArray[1].commands[19].valueFlags[1..4].flagMode := 1;
   // movePath.pathDataArray[1].commands[20].valueFlags[1..4].flagMode := 1;
   // movePath.pathDataArray[2].commands[1].valueFlags[1..4].flagMode := 1;
   // movePath.pathDataArray[2].commands[2].valueFlags[1..4].flagMode := 1;
   // movePath.pathDataArray[2].commands[3].valueFlags[1..4].flagMode := 1;
   // movePath.pathDataArray[2].commands[4].valueFlags[1..4].flagMode := 1;
   // movePath.pathDataArray[2].commands[5].valueFlags[1..4].flagMode := 1;
   // movePath.pathDataArray[2].commands[6].valueFlags[1..4].flagMode := 1;
   // movePath.pathDataArray[2].commands[7].valueFlags[1..4].flagMode := 1;
   // movePath.pathDataArray[2].commands[8].valueFlags[1..4].flagMode := 1;
   // movePath.pathDataArray[2].commands[9].valueFlags[1..4].flagMode := 1;
   // movePath.pathDataArray[2].commands[10].valueFlags[1..4].flagMode := 1;
   // movePath.pathDataArray[2].commands[11].valueFlags[1..4].flagMode := 1;
   // movePath.pathDataArray[2].commands[12].valueFlags[1..4].flagMode := 1;
   // movePath.pathDataArray[2].commands[13].valueFlags[1..4].flagMode := 1;
   // movePath.pathDataArray[2].commands[14].valueFlags[1..4].flagMode := 1;
   // movePath.pathDataArray[2].commands[15].valueFlags[1..4].flagMode := 1;
   // movePath.pathDataArray[2].commands[16].valueFlags[1..4].flagMode := 1;
   // movePath.pathDataArray[2].commands[17].valueFlags[1..4].flagMode := 1;
   // movePath.pathDataArray[2].commands[18].valueFlags[1..4].flagMode := 1;
   // movePath.pathDataArray[2].commands[19].valueFlags[1..4].flagMode := 1;
   // movePath.pathDataArray[2].commands[20].valueFlags[1..4].flagMode := 1;
   // movePath.pathDataArray[3].commands[1].valueFlags[1..4].flagMode := 1;
   // movePath.pathDataArray[3].commands[2].valueFlags[1..4].flagMode := 1;
   // movePath.pathDataArray[3].commands[3].valueFlags[1..4].flagMode := 1;
   // movePath.pathDataArray[3].commands[4].valueFlags[1..4].flagMode := 1;
   // movePath.pathDataArray[3].commands[5].valueFlags[1..4].flagMode := 1;
   // movePath.pathDataArray[3].commands[6].valueFlags[1..4].flagMode := 1;
   // movePath.pathDataArray[3].commands[7].valueFlags[1..4].flagMode := 1;
   // movePath.pathDataArray[3].commands[8].valueFlags[1..4].flagMode := 1;
   // movePath.pathDataArray[3].commands[9].valueFlags[1..4].flagMode := 1;
   // movePath.pathDataArray[3].commands[10].valueFlags[1..4].flagMode := 1;
   // movePath.pathDataArray[3].commands[11].valueFlags[1..4].flagMode := 1;
   // movePath.pathDataArray[3].commands[12].valueFlags[1..4].flagMode := 1;
   // movePath.pathDataArray[3].commands[13].valueFlags[1..4].flagMode := 1;
   // movePath.pathDataArray[3].commands[14].valueFlags[1..4].flagMode := 1;
   // movePath.pathDataArray[3].commands[15].valueFlags[1..4].flagMode := 1;
   // movePath.pathDataArray[3].commands[16].valueFlags[1..4].flagMode := 1;
   // movePath.pathDataArray[3].commands[17].valueFlags[1..4].flagMode := 1;
   // movePath.pathDataArray[3].commands[18].valueFlags[1..4].flagMode := 1;
   // movePath.pathDataArray[3].commands[19].valueFlags[1..4].flagMode := 1;
   // movePath.pathDataArray[3].commands[20].valueFlags[1..4].flagMode := 1;
   // movePath.pathDataArray[4].commands[1].valueFlags[1..4].flagMode := 1;
   // movePath.pathDataArray[4].commands[2].valueFlags[1..4].flagMode := 1;
   // movePath.pathDataArray[4].commands[3].valueFlags[1..4].flagMode := 1;
   // movePath.pathDataArray[4].commands[4].valueFlags[1..4].flagMode := 1;
   // movePath.pathDataArray[4].commands[5].valueFlags[1..4].flagMode := 1;
   // movePath.pathDataArray[4].commands[6].valueFlags[1..4].flagMode := 1;
   // movePath.pathDataArray[4].commands[7].valueFlags[1..4].flagMode := 1;
   // movePath.pathDataArray[4].commands[8].valueFlags[1..4].flagMode := 1;
   // movePath.pathDataArray[4].commands[9].valueFlags[1..4].flagMode := 1;
   // movePath.pathDataArray[4].commands[10].valueFlags[1..4].flagMode := 1;
   // movePath.pathDataArray[4].commands[11].valueFlags[1..4].flagMode := 1;
   // movePath.pathDataArray[4].commands[12].valueFlags[1..4].flagMode := 1;
   // movePath.pathDataArray[4].commands[13].valueFlags[1..4].flagMode := 1;
   // movePath.pathDataArray[4].commands[14].valueFlags[1..4].flagMode := 1;
   // movePath.pathDataArray[4].commands[15].valueFlags[1..4].flagMode := 1;
   // movePath.pathDataArray[4].commands[16].valueFlags[1..4].flagMode := 1;
   // movePath.pathDataArray[4].commands[17].valueFlags[1..4].flagMode := 1;
   // movePath.pathDataArray[4].commands[18].valueFlags[1..4].flagMode := 1;
   // movePath.pathDataArray[4].commands[19].valueFlags[1..4].flagMode := 1;
   // movePath.pathDataArray[4].commands[20].valueFlags[1..4].flagMode := 1;
   // movePath.pathDataArray[5].commands[1].valueFlags[1..4].flagMode := 1;
   // movePath.pathDataArray[5].commands[2].valueFlags[1..4].flagMode := 1;
   // movePath.pathDataArray[5].commands[3].valueFlags[1..4].flagMode := 1;
   // movePath.pathDataArray[5].commands[4].valueFlags[1..4].flagMode := 1;
   // movePath.pathDataArray[5].commands[5].valueFlags[1..4].flagMode := 1;
   // movePath.pathDataArray[5].commands[6].valueFlags[1..4].flagMode := 1;
   // movePath.pathDataArray[5].commands[7].valueFlags[1..4].flagMode := 1;
   // movePath.pathDataArray[5].commands[8].valueFlags[1..4].flagMode := 1;
   // movePath.pathDataArray[5].commands[9].valueFlags[1..4].flagMode := 1;
   // movePath.pathDataArray[5].commands[10].valueFlags[1..4].flagMode := 1;
   // movePath.pathDataArray[5].commands[11].valueFlags[1..4].flagMode := 1;
   // movePath.pathDataArray[5].commands[12].valueFlags[1..4].flagMode := 1;
   // movePath.pathDataArray[5].commands[13].valueFlags[1..4].flagMode := 1;
   // movePath.pathDataArray[5].commands[14].valueFlags[1..4].flagMode := 1;
   // movePath.pathDataArray[5].commands[15].valueFlags[1..4].flagMode := 1;
   // movePath.pathDataArray[5].commands[16].valueFlags[1..4].flagMode := 1;
   // movePath.pathDataArray[5].commands[17].valueFlags[1..4].flagMode := 1;
   // movePath.pathDataArray[5].commands[18].valueFlags[1..4].flagMode := 1;
   // movePath.pathDataArray[5].commands[19].valueFlags[1..4].flagMode := 1;
   // movePath.pathDataArray[5].commands[20].valueFlags[1..4].flagMode := 1;
   // movePath.pathDataArray[1].commands[1].valueFlags[1..4].remainingDistance := -1.0;
   // movePath.pathDataArray[1].commands[2].valueFlags[1..4].remainingDistance := -1.0;
   // movePath.pathDataArray[1].commands[3].valueFlags[1..4].remainingDistance := -1.0;
   // movePath.pathDataArray[1].commands[4].valueFlags[1..4].remainingDistance := -1.0;
   // movePath.pathDataArray[1].commands[5].valueFlags[1..4].remainingDistance := -1.0;
   // movePath.pathDataArray[1].commands[6].valueFlags[1..4].remainingDistance := -1.0;
   // movePath.pathDataArray[1].commands[7].valueFlags[1..4].remainingDistance := -1.0;
   // movePath.pathDataArray[1].commands[8].valueFlags[1..4].remainingDistance := -1.0;
   // movePath.pathDataArray[1].commands[9].valueFlags[1..4].remainingDistance := -1.0;
   // movePath.pathDataArray[1].commands[10].valueFlags[1..4].remainingDistance := 0.0;
   // movePath.pathDataArray[1].commands[11].valueFlags[1..4].remainingDistance := -1.0;
   // movePath.pathDataArray[1].commands[12].valueFlags[1..4].remainingDistance := -1.0;
   // movePath.pathDataArray[1].commands[13].valueFlags[1..4].remainingDistance := -1.0;
   // movePath.pathDataArray[1].commands[14].valueFlags[1..4].remainingDistance := -1.0;
   // movePath.pathDataArray[1].commands[15].valueFlags[1..4].remainingDistance := -1.0;
   // movePath.pathDataArray[1].commands[16].valueFlags[1..4].remainingDistance := -1.0;
   // movePath.pathDataArray[1].commands[17].valueFlags[1..4].remainingDistance := -1.0;
   // movePath.pathDataArray[1].commands[18].valueFlags[1..4].remainingDistance := -1.0;
   // movePath.pathDataArray[1].commands[19].valueFlags[1..4].remainingDistance := -1.0;
   // movePath.pathDataArray[1].commands[20].valueFlags[1..4].remainingDistance := -1.0;
   // movePath.pathDataArray[2].commands[1].valueFlags[1..4].remainingDistance := -1.0;
   // movePath.pathDataArray[2].commands[2].valueFlags[1..4].remainingDistance := -1.0;
   // movePath.pathDataArray[2].commands[3].valueFlags[1..4].remainingDistance := -1.0;
   // movePath.pathDataArray[2].commands[4].valueFlags[1..4].remainingDistance := -1.0;
   // movePath.pathDataArray[2].commands[5].valueFlags[1..4].remainingDistance := -1.0;
   // movePath.pathDataArray[2].commands[6].valueFlags[1..4].remainingDistance := -1.0;
   // movePath.pathDataArray[2].commands[7].valueFlags[1..4].remainingDistance := -1.0;
   // movePath.pathDataArray[2].commands[8].valueFlags[1..4].remainingDistance := -1.0;
   // movePath.pathDataArray[2].commands[9].valueFlags[1..4].remainingDistance := -1.0;
   // movePath.pathDataArray[2].commands[10].valueFlags[1..4].remainingDistance := -1.0;
   // movePath.pathDataArray[2].commands[11].valueFlags[1..4].remainingDistance := 0.0;
   // movePath.pathDataArray[2].commands[12].valueFlags[1..4].remainingDistance := -1.0;
   // movePath.pathDataArray[2].commands[13].valueFlags[1..4].remainingDistance := -1.0;
   // movePath.pathDataArray[2].commands[14].valueFlags[1..4].remainingDistance := -1.0;
   // movePath.pathDataArray[2].commands[15].valueFlags[1..4].remainingDistance := -1.0;
   // movePath.pathDataArray[2].commands[16].valueFlags[1..4].remainingDistance := -1.0;
   // movePath.pathDataArray[2].commands[17].valueFlags[1..4].remainingDistance := -1.0;
   // movePath.pathDataArray[2].commands[18].valueFlags[1..4].remainingDistance := -1.0;
   // movePath.pathDataArray[2].commands[19].valueFlags[1..4].remainingDistance := -1.0;
   // movePath.pathDataArray[2].commands[20].valueFlags[1..4].remainingDistance := -1.0;
   // movePath.pathDataArray[3].commands[1].valueFlags[1..4].remainingDistance := -1.0;
   // movePath.pathDataArray[3].commands[2].valueFlags[1..4].remainingDistance := -1.0;
   // movePath.pathDataArray[3].commands[3].valueFlags[1..4].remainingDistance := -1.0;
   // movePath.pathDataArray[3].commands[4].valueFlags[1..4].remainingDistance := -1.0;
   // movePath.pathDataArray[3].commands[5].valueFlags[1..4].remainingDistance := -1.0;
   // movePath.pathDataArray[3].commands[6].valueFlags[1..4].remainingDistance := -1.0;
   // movePath.pathDataArray[3].commands[7].valueFlags[1..4].remainingDistance := -1.0;
   // movePath.pathDataArray[3].commands[8].valueFlags[1..4].remainingDistance := -1.0;
   // movePath.pathDataArray[3].commands[9].valueFlags[1..4].remainingDistance := -1.0;
   // movePath.pathDataArray[3].commands[10].valueFlags[1..4].remainingDistance := -1.0;
   // movePath.pathDataArray[3].commands[11].valueFlags[1..4].remainingDistance := -1.0;
   // movePath.pathDataArray[3].commands[12].valueFlags[1..4].remainingDistance := -1.0;
   // movePath.pathDataArray[3].commands[13].valueFlags[1..4].remainingDistance := -1.0;
   // movePath.pathDataArray[3].commands[14].valueFlags[1..4].remainingDistance := -1.0;
   // movePath.pathDataArray[3].commands[15].valueFlags[1..4].remainingDistance := -1.0;
   // movePath.pathDataArray[3].commands[16].valueFlags[1..4].remainingDistance := -1.0;
   // movePath.pathDataArray[3].commands[17].valueFlags[1..4].remainingDistance := -1.0;
   // movePath.pathDataArray[3].commands[18].valueFlags[1..4].remainingDistance := -1.0;
   // movePath.pathDataArray[3].commands[19].valueFlags[1..4].remainingDistance := -1.0;
   // movePath.pathDataArray[3].commands[20].valueFlags[1..4].remainingDistance := -1.0;
   // movePath.pathDataArray[4].commands[1].valueFlags[1..4].remainingDistance := -1.0;
   // movePath.pathDataArray[4].commands[2].valueFlags[1..4].remainingDistance := -1.0;
   // movePath.pathDataArray[4].commands[3].valueFlags[1..4].remainingDistance := -1.0;
   // movePath.pathDataArray[4].commands[4].valueFlags[1..4].remainingDistance := -1.0;
   // movePath.pathDataArray[4].commands[5].valueFlags[1..4].remainingDistance := -1.0;
   // movePath.pathDataArray[4].commands[6].valueFlags[1..4].remainingDistance := -1.0;
   // movePath.pathDataArray[4].commands[7].valueFlags[1..4].remainingDistance := -1.0;
   // movePath.pathDataArray[4].commands[8].valueFlags[1..4].remainingDistance := -1.0;
   // movePath.pathDataArray[4].commands[9].valueFlags[1..4].remainingDistance := -1.0;
   // movePath.pathDataArray[4].commands[10].valueFlags[1..4].remainingDistance := -1.0;
   // movePath.pathDataArray[4].commands[11].valueFlags[1..4].remainingDistance := -1.0;
   // movePath.pathDataArray[4].commands[12].valueFlags[1..4].remainingDistance := -1.0;
   // movePath.pathDataArray[4].commands[13].valueFlags[1..4].remainingDistance := -1.0;
   // movePath.pathDataArray[4].commands[14].valueFlags[1..4].remainingDistance := -1.0;
   // movePath.pathDataArray[4].commands[15].valueFlags[1..4].remainingDistance := -1.0;
   // movePath.pathDataArray[4].commands[16].valueFlags[1..4].remainingDistance := -1.0;
   // movePath.pathDataArray[4].commands[17].valueFlags[1..4].remainingDistance := -1.0;
   // movePath.pathDataArray[4].commands[18].valueFlags[1..4].remainingDistance := -1.0;
   // movePath.pathDataArray[4].commands[19].valueFlags[1..4].remainingDistance := -1.0;
   // movePath.pathDataArray[4].commands[20].valueFlags[1..4].remainingDistance := -1.0;
   // movePath.pathDataArray[5].commands[1].valueFlags[1..4].remainingDistance := -1.0;
   // movePath.pathDataArray[5].commands[2].valueFlags[1..4].remainingDistance := -1.0;
   // movePath.pathDataArray[5].commands[3].valueFlags[1..4].remainingDistance := -1.0;
   // movePath.pathDataArray[5].commands[4].valueFlags[1..4].remainingDistance := -1.0;
   // movePath.pathDataArray[5].commands[5].valueFlags[1..4].remainingDistance := -1.0;
   // movePath.pathDataArray[5].commands[6].valueFlags[1..4].remainingDistance := -1.0;
   // movePath.pathDataArray[5].commands[7].valueFlags[1..4].remainingDistance := -1.0;
   // movePath.pathDataArray[5].commands[8].valueFlags[1..4].remainingDistance := -1.0;
   // movePath.pathDataArray[5].commands[9].valueFlags[1..4].remainingDistance := -1.0;
   // movePath.pathDataArray[5].commands[10].valueFlags[1..4].remainingDistance := -1.0;
   // movePath.pathDataArray[5].commands[11].valueFlags[1..4].remainingDistance := -1.0;
   // movePath.pathDataArray[5].commands[12].valueFlags[1..4].remainingDistance := -1.0;
   // movePath.pathDataArray[5].commands[13].valueFlags[1..4].remainingDistance := -1.0;
   // movePath.pathDataArray[5].commands[14].valueFlags[1..4].remainingDistance := -1.0;
   // movePath.pathDataArray[5].commands[15].valueFlags[1..4].remainingDistance := -1.0;
   // movePath.pathDataArray[5].commands[16].valueFlags[1..4].remainingDistance := -1.0;
   // movePath.pathDataArray[5].commands[17].valueFlags[1..4].remainingDistance := -1.0;
   // movePath.pathDataArray[5].commands[18].valueFlags[1..4].remainingDistance := -1.0;
   // movePath.pathDataArray[5].commands[19].valueFlags[1..4].remainingDistance := -1.0;
   // movePath.pathDataArray[5].commands[20].valueFlags[1..4].remainingDistance := -1.0;
   // movePath.pathDataArray[1].commands[1].parameterValid[1..6] := TRUE;
   // movePath.pathDataArray[1].commands[2].parameterValid[1..6] := TRUE;
   // movePath.pathDataArray[1].commands[3].parameterValid[1..6] := TRUE;
   // movePath.pathDataArray[1].commands[4].parameterValid[1..6] := TRUE;
   // movePath.pathDataArray[1].commands[5].parameterValid[1..6] := TRUE;
   // movePath.pathDataArray[1].commands[6].parameterValid[1..6] := TRUE;
   // movePath.pathDataArray[1].commands[7].parameterValid[1..6] := TRUE;
   // movePath.pathDataArray[1].commands[8].parameterValid[1..6] := TRUE;
   // movePath.pathDataArray[1].commands[9].parameterValid[1..6] := TRUE;
   // movePath.pathDataArray[1].commands[10].parameterValid[1..6] := TRUE;
   // movePath.pathDataArray[1].commands[11].parameterValid[1..6] := TRUE;
   // movePath.pathDataArray[1].commands[12].parameterValid[1..6] := TRUE;
   // movePath.pathDataArray[1].commands[13].parameterValid[1..6] := TRUE;
   // movePath.pathDataArray[1].commands[14].parameterValid[1..6] := TRUE;
   // movePath.pathDataArray[1].commands[15].parameterValid[1..6] := TRUE;
   // movePath.pathDataArray[1].commands[16].parameterValid[1..6] := TRUE;
   // movePath.pathDataArray[1].commands[17].parameterValid[1..6] := TRUE;
   // movePath.pathDataArray[1].commands[18].parameterValid[1..6] := TRUE;
   // movePath.pathDataArray[1].commands[19].parameterValid[1..6] := TRUE;
   // movePath.pathDataArray[1].commands[20].parameterValid[1..6] := TRUE;
   // movePath.pathDataArray[2].commands[1].parameterValid[1..6] := TRUE;
   // movePath.pathDataArray[2].commands[2].parameterValid[1..6] := TRUE;
   // movePath.pathDataArray[2].commands[3].parameterValid[1..6] := TRUE;
   // movePath.pathDataArray[2].commands[4].parameterValid[1..6] := TRUE;
   // movePath.pathDataArray[2].commands[5].parameterValid[1..6] := TRUE;
   // movePath.pathDataArray[2].commands[6].parameterValid[1..6] := TRUE;
   // movePath.pathDataArray[2].commands[7].parameterValid[1..6] := TRUE;
   // movePath.pathDataArray[2].commands[8].parameterValid[1..6] := TRUE;
   // movePath.pathDataArray[2].commands[9].parameterValid[1..6] := TRUE;
   // movePath.pathDataArray[2].commands[10].parameterValid[1..6] := TRUE;
   // movePath.pathDataArray[2].commands[11].parameterValid[1..6] := TRUE;
   // movePath.pathDataArray[2].commands[12].parameterValid[1..6] := TRUE;
   // movePath.pathDataArray[2].commands[13].parameterValid[1..6] := TRUE;
   // movePath.pathDataArray[2].commands[14].parameterValid[1..6] := TRUE;
   // movePath.pathDataArray[2].commands[15].parameterValid[1..6] := TRUE;
   // movePath.pathDataArray[2].commands[16].parameterValid[1..6] := TRUE;
   // movePath.pathDataArray[2].commands[17].parameterValid[1..6] := TRUE;
   // movePath.pathDataArray[2].commands[18].parameterValid[1..6] := TRUE;
   // movePath.pathDataArray[2].commands[19].parameterValid[1..6] := TRUE;
   // movePath.pathDataArray[2].commands[20].parameterValid[1..6] := TRUE;
   // movePath.pathDataArray[3].commands[1].parameterValid[1..6] := TRUE;
   // movePath.pathDataArray[3].commands[2].parameterValid[1..6] := TRUE;
   // movePath.pathDataArray[3].commands[3].parameterValid[1..6] := TRUE;
   // movePath.pathDataArray[3].commands[4].parameterValid[1..6] := TRUE;
   // movePath.pathDataArray[3].commands[5].parameterValid[1..6] := TRUE;
   // movePath.pathDataArray[3].commands[6].parameterValid[1..6] := TRUE;
   // movePath.pathDataArray[3].commands[7].parameterValid[1..6] := TRUE;
   // movePath.pathDataArray[3].commands[8].parameterValid[1..6] := TRUE;
   // movePath.pathDataArray[3].commands[9].parameterValid[1..6] := TRUE;
   // movePath.pathDataArray[3].commands[10].parameterValid[1..6] := TRUE;
   // movePath.pathDataArray[3].commands[11].parameterValid[1..6] := TRUE;
   // movePath.pathDataArray[3].commands[12].parameterValid[1..6] := TRUE;
   // movePath.pathDataArray[3].commands[13].parameterValid[1..6] := TRUE;
   // movePath.pathDataArray[3].commands[14].parameterValid[1..6] := TRUE;
   // movePath.pathDataArray[3].commands[15].parameterValid[1..6] := TRUE;
   // movePath.pathDataArray[3].commands[16].parameterValid[1..6] := TRUE;
   // movePath.pathDataArray[3].commands[17].parameterValid[1..6] := TRUE;
   // movePath.pathDataArray[3].commands[18].parameterValid[1..6] := TRUE;
   // movePath.pathDataArray[3].commands[19].parameterValid[1..6] := TRUE;
   // movePath.pathDataArray[3].commands[20].parameterValid[1..6] := TRUE;
   // movePath.pathDataArray[4].commands[1].parameterValid[1..6] := TRUE;
   // movePath.pathDataArray[4].commands[2].parameterValid[1..6] := TRUE;
   // movePath.pathDataArray[4].commands[3].parameterValid[1..6] := TRUE;
   // movePath.pathDataArray[4].commands[4].parameterValid[1..6] := TRUE;
   // movePath.pathDataArray[4].commands[5].parameterValid[1..6] := TRUE;
   // movePath.pathDataArray[4].commands[6].parameterValid[1..6] := TRUE;
   // movePath.pathDataArray[4].commands[7].parameterValid[1..6] := TRUE;
   // movePath.pathDataArray[4].commands[8].parameterValid[1..6] := TRUE;
   // movePath.pathDataArray[4].commands[9].parameterValid[1..6] := TRUE;
   // movePath.pathDataArray[4].commands[10].parameterValid[1..6] := TRUE;
   // movePath.pathDataArray[4].commands[11].parameterValid[1..6] := TRUE;
   // movePath.pathDataArray[4].commands[12].parameterValid[1..6] := TRUE;
   // movePath.pathDataArray[4].commands[13].parameterValid[1..6] := TRUE;
   // movePath.pathDataArray[4].commands[14].parameterValid[1..6] := TRUE;
   // movePath.pathDataArray[4].commands[15].parameterValid[1..6] := TRUE;
   // movePath.pathDataArray[4].commands[16].parameterValid[1..6] := TRUE;
   // movePath.pathDataArray[4].commands[17].parameterValid[1..6] := TRUE;
   // movePath.pathDataArray[4].commands[18].parameterValid[1..6] := TRUE;
   // movePath.pathDataArray[4].commands[19].parameterValid[1..6] := TRUE;
   // movePath.pathDataArray[4].commands[20].parameterValid[1..6] := TRUE;
   // movePath.pathDataArray[5].commands[1].parameterValid[1..6] := TRUE;
   // movePath.pathDataArray[5].commands[2].parameterValid[1..6] := TRUE;
   // movePath.pathDataArray[5].commands[3].parameterValid[1..6] := TRUE;
   // movePath.pathDataArray[5].commands[4].parameterValid[1..6] := TRUE;
   // movePath.pathDataArray[5].commands[5].parameterValid[1..6] := TRUE;
   // movePath.pathDataArray[5].commands[6].parameterValid[1..6] := TRUE;
   // movePath.pathDataArray[5].commands[7].parameterValid[1..6] := TRUE;
   // movePath.pathDataArray[5].commands[8].parameterValid[1..6] := TRUE;
   // movePath.pathDataArray[5].commands[9].parameterValid[1..6] := TRUE;
   // movePath.pathDataArray[5].commands[10].parameterValid[1..6] := TRUE;
   // movePath.pathDataArray[5].commands[11].parameterValid[1..6] := TRUE;
   // movePath.pathDataArray[5].commands[12].parameterValid[1..6] := TRUE;
   // movePath.pathDataArray[5].commands[13].parameterValid[1..6] := TRUE;
   // movePath.pathDataArray[5].commands[14].parameterValid[1..6] := TRUE;
   // movePath.pathDataArray[5].commands[15].parameterValid[1..6] := TRUE;
   // movePath.pathDataArray[5].commands[16].parameterValid[1..6] := TRUE;
   // movePath.pathDataArray[5].commands[17].parameterValid[1..6] := TRUE;
   // movePath.pathDataArray[5].commands[18].parameterValid[1..6] := TRUE;
   // movePath.pathDataArray[5].commands[19].parameterValid[1..6] := TRUE;
   // movePath.pathDataArray[5].commands[20].parameterValid[1..6] := TRUE;
   // movePath.pointTable[1]."name" := WSTRING#'S2 Above place';
   // movePath.pointTable[2]."name" := WSTRING#'S2 Place';
   // movePath.pointTable[3..30]."name" := WSTRING#'- - -';
   // movePath.pointTable[1].position[0..1] := 0.0;
   // movePath.pointTable[1].position[2] := 30.0;
   // movePath.pointTable[1].position[3] := 90.0;
   // movePath.pointTable[1].position[4..5] := 0.0;
   // movePath.pointTable[2].position[0..2] := 0.0;
   // movePath.pointTable[2].position[3] := 90.0;
   // movePath.pointTable[2].position[4..5] := 0.0;
   // movePath.pointTable[3].position[0..5] := 0.0;
   // movePath.pointTable[4].position[0..5] := 0.0;
   // movePath.pointTable[5].position[0..5] := 0.0;
   // movePath.pointTable[6].position[0..5] := 0.0;
   // movePath.pointTable[7].position[0..5] := 0.0;
   // movePath.pointTable[8].position[0..5] := 0.0;
   // movePath.pointTable[9].position[0..5] := 0.0;
   // movePath.pointTable[10].position[0..5] := 0.0;
   // movePath.pointTable[11].position[0..5] := 0.0;
   // movePath.pointTable[12].position[0..5] := 0.0;
   // movePath.pointTable[13].position[0..5] := 0.0;
   // movePath.pointTable[14].position[0..5] := 0.0;
   // movePath.pointTable[15].position[0..5] := 0.0;
   // movePath.pointTable[16].position[0..5] := 0.0;
   // movePath.pointTable[17].position[0..5] := 0.0;
   // movePath.pointTable[18].position[0..5] := 0.0;
   // movePath.pointTable[19].position[0..5] := 0.0;
   // movePath.pointTable[20].position[0..5] := 0.0;
   // movePath.pointTable[21].position[0..5] := 0.0;
   // movePath.pointTable[22].position[0..5] := 0.0;
   // movePath.pointTable[23].position[0..5] := 0.0;
   // movePath.pointTable[24].position[0..5] := 0.0;
   // movePath.pointTable[25].position[0..5] := 0.0;
   // movePath.pointTable[26].position[0..5] := 0.0;
   // movePath.pointTable[27].position[0..5] := 0.0;
   // movePath.pointTable[28].position[0..5] := 0.0;
   // movePath.pointTable[29].position[0..5] := 0.0;
   // movePath.pointTable[30].position[0..5] := 0.0;
   // movePath.pointTable[1..2].coordSystem := 11;
   // movePath.pointTable[3..30].coordSystem := 0;
   // movePath.pointTable[1..30].linkConstellation := 16#FFFF_FFFF;
   // movePath.pointTable[1].turnJoint[0..5] := 0;
   // movePath.pointTable[2].turnJoint[0..5] := 0;
   // movePath.pointTable[3].turnJoint[0..5] := 0;
   // movePath.pointTable[4].turnJoint[0..5] := 0;
   // movePath.pointTable[5].turnJoint[0..5] := 0;
   // movePath.pointTable[6].turnJoint[0..5] := 0;
   // movePath.pointTable[7].turnJoint[0..5] := 0;
   // movePath.pointTable[8].turnJoint[0..5] := 0;
   // movePath.pointTable[9].turnJoint[0..5] := 0;
   // movePath.pointTable[10].turnJoint[0..5] := 0;
   // movePath.pointTable[11].turnJoint[0..5] := 0;
   // movePath.pointTable[12].turnJoint[0..5] := 0;
   // movePath.pointTable[13].turnJoint[0..5] := 0;
   // movePath.pointTable[14].turnJoint[0..5] := 0;
   // movePath.pointTable[15].turnJoint[0..5] := 0;
   // movePath.pointTable[16].turnJoint[0..5] := 0;
   // movePath.pointTable[17].turnJoint[0..5] := 0;
   // movePath.pointTable[18].turnJoint[0..5] := 0;
   // movePath.pointTable[19].turnJoint[0..5] := 0;
   // movePath.pointTable[20].turnJoint[0..5] := 0;
   // movePath.pointTable[21].turnJoint[0..5] := 0;
   // movePath.pointTable[22].turnJoint[0..5] := 0;
   // movePath.pointTable[23].turnJoint[0..5] := 0;
   // movePath.pointTable[24].turnJoint[0..5] := 0;
   // movePath.pointTable[25].turnJoint[0..5] := 0;
   // movePath.pointTable[26].turnJoint[0..5] := 0;
   // movePath.pointTable[27].turnJoint[0..5] := 0;
   // movePath.pointTable[28].turnJoint[0..5] := 0;
   // movePath.pointTable[29].turnJoint[0..5] := 0;
   // movePath.pointTable[30].turnJoint[0..5] := 0;
   // movePath.setFlagNames[0] := WSTRING#'S1 Enable actuator';
   // movePath.setFlagNames[1] := WSTRING#'S1 Disable actuator';
   // movePath.setFlagNames[2] := WSTRING#'S2 Pick ready';
   // movePath.setFlagNames[3] := WSTRING#'S2 Open actuator';
   // movePath.setFlagNames[4] := WSTRING#'S2 Close actuator';
   // movePath.setFlagNames[5] := WSTRING#'S3 Product detected conveyor 1';
   // movePath.setFlagNames[6..30] := WSTRING#'- - -';
   // movePath.valueFlagNames[0..30] := WSTRING#'- - -';
   // movePath.settings.kinematics."name" := WSTRING#'Rollpicker';
   // movePath.settings.kinematics.jogPath.accelerationTime := 0.2;
   // movePath.settings.kinematics.jogPath.maxVelocityManual := 250.0;
   // movePath.settings.kinematics.jogPath.maxVelocityTestRun := 250.0;
   // movePath.settings.kinematics.jogPath.presetIncrementCoarse := 10.0;
   // movePath.settings.kinematics.jogPath.presetIncrementFine := 1.0;
   // movePath.settings.kinematics.jogPath.presetIncrementPrecise := 0.1;
   // movePath.settings.kinematics.jogOrientation.accelerationTime := 0.2;
   // movePath.settings.kinematics.jogOrientation.maxVelocityManual := 30.0;
   // movePath.settings.kinematics.jogOrientation.maxVelocityTestRun := 45.0;
   // movePath.settings.kinematics.jogOrientation.presetIncrementCoarse := 5.0;
   // movePath.settings.kinematics.jogOrientation.presetIncrementFine := 1.0;
   // movePath.settings.kinematics.jogOrientation.presetIncrementPrecise := 0.1;
   // movePath.settings.kinematicAxes[1]."name" := WSTRING#'KinAxis A1';
   // movePath.settings.kinematicAxes[2]."name" := WSTRING#'KinAxis A2';
   // movePath.settings.kinematicAxes[3]."name" := WSTRING#'KinAxis A3';
   // movePath.settings.kinematicAxes[4]."name" := WSTRING#'KinAxis A4';
   // movePath.settings.kinematicAxes[5]."name" := WSTRING#'KinAxis A5';
   // movePath.settings.kinematicAxes[6]."name" := WSTRING#'KinAxis A6';
   // movePath.settings.kinematicAxes[1..6].used := FALSE;
   // movePath.settings.kinematicAxes[1..6].withBrake := FALSE;
   // movePath.settings.kinematicAxes[1..6].homePosition := 0.0;
   // movePath.settings.kinematicAxes[1..6].coupling := FALSE;
   // movePath.settings.kinematicAxes[1..6].jog.accelerationTime := 0.2;
   // movePath.settings.kinematicAxes[1..2].jog.maxVelocityManual := 200.0;
   // movePath.settings.kinematicAxes[3].jog.maxVelocityManual := 250.0;
   // movePath.settings.kinematicAxes[4].jog.maxVelocityManual := 30.0;
   // movePath.settings.kinematicAxes[5..6].jog.maxVelocityManual := 10.0;
   // movePath.settings.kinematicAxes[1..3].jog.maxVelocityTestRun := 250.0;
   // movePath.settings.kinematicAxes[4].jog.maxVelocityTestRun := 45.0;
   // movePath.settings.kinematicAxes[5..6].jog.maxVelocityTestRun := 10.0;
   // movePath.settings.kinematicAxes[1..2].jog.presetIncrementCoarse := 5.0;
   // movePath.settings.kinematicAxes[3].jog.presetIncrementCoarse := 10.0;
   // movePath.settings.kinematicAxes[4..6].jog.presetIncrementCoarse := 5.0;
   // movePath.settings.kinematicAxes[1..2].jog.presetIncrementFine := 1.0;
   // movePath.settings.kinematicAxes[3].jog.presetIncrementFine := 5.0;
   // movePath.settings.kinematicAxes[4..6].jog.presetIncrementFine := 1.0;
   // movePath.settings.kinematicAxes[1..2].jog.presetIncrementPrecise := 0.5;
   // movePath.settings.kinematicAxes[3].jog.presetIncrementPrecise := 0.1;
   // movePath.settings.kinematicAxes[4..6].jog.presetIncrementPrecise := 0.5;
   // movePath.settings.movePathConfiguration.offsetParameter[1..3]."name" := '- - -';
   // movePath.settings.movePathConfiguration.offsetParameter[1..3].radius := 0.0;
   // movePath.settings.movePathConfiguration.offsetParameter[1..3].length := 0.0;
   // movePath.settings.movePathConfiguration.conveyorParameter[1].conveyorBeltAxis := 28;
   // movePath.settings.movePathConfiguration.conveyorParameter[2].conveyorBeltAxis := 27;
   // movePath.settings.movePathConfiguration.conveyorParameter[3..5].conveyorBeltAxis := 0;
   // movePath.settings.movePathConfiguration.conveyorParameter[1].conveyorBeltOrigin.x := 0.0;
   // movePath.settings.movePathConfiguration.conveyorParameter[2].conveyorBeltOrigin.x := 300.0;
   // movePath.settings.movePathConfiguration.conveyorParameter[3..5].conveyorBeltOrigin.x := 0.0;
   // movePath.settings.movePathConfiguration.conveyorParameter[1].conveyorBeltOrigin.y := 50.0;
   // movePath.settings.movePathConfiguration.conveyorParameter[2].conveyorBeltOrigin.y := -100.0;
   // movePath.settings.movePathConfiguration.conveyorParameter[3..5].conveyorBeltOrigin.y := 0.0;
   // movePath.settings.movePathConfiguration.conveyorParameter[1..5].conveyorBeltOrigin.z := 0.0;
   // movePath.settings.movePathConfiguration.conveyorParameter[1].conveyorBeltOrigin."a" := 0.0;
   // movePath.settings.movePathConfiguration.conveyorParameter[2].conveyorBeltOrigin."a" := -180.0;
   // movePath.settings.movePathConfiguration.conveyorParameter[3..5].conveyorBeltOrigin."a" := 0.0;
   // movePath.settings.movePathConfiguration.conveyorParameter[1..5].conveyorBeltOrigin."b" := 0.0;
   // movePath.settings.movePathConfiguration.conveyorParameter[1..5].conveyorBeltOrigin.c := 0.0;
   // movePath.settings.movePathConfiguration.conveyorParameter[1].initialObjectPosition.x := 420.018;
   // movePath.settings.movePathConfiguration.conveyorParameter[2].initialObjectPosition.x := 550.44;
   // movePath.settings.movePathConfiguration.conveyorParameter[3..5].initialObjectPosition.x := 0.0;
   // movePath.settings.movePathConfiguration.conveyorParameter[1..5].initialObjectPosition.y := 0.0;
   // movePath.settings.movePathConfiguration.conveyorParameter[1..5].initialObjectPosition.z := 0.0;
   // movePath.settings.movePathConfiguration.conveyorParameter[1..5].initialObjectPosition."a" := 0.0;
   // movePath.settings.movePathConfiguration.conveyorParameter[1..5].initialObjectPosition."b" := 0.0;
   // movePath.settings.movePathConfiguration.conveyorParameter[1..5].initialObjectPosition.c := 0.0;
   // movePath.settings.movePathConfiguration.userFrames[11].x := 100.0;
   // movePath.settings.movePathConfiguration.userFrames[12..15].x := 0.0;
   // movePath.settings.movePathConfiguration.userFrames[11].y := 200.0;
   // movePath.settings.movePathConfiguration.userFrames[12..15].y := 0.0;
   // movePath.settings.movePathConfiguration.userFrames[11].z := 20.0;
   // movePath.settings.movePathConfiguration.userFrames[12..15].z := 0.0;
   // movePath.settings.movePathConfiguration.userFrames[11..15]."a" := 0.0;
   // movePath.settings.movePathConfiguration.userFrames[11..15]."b" := 0.0;
   // movePath.settings.movePathConfiguration.userFrames[11..15].c := 0.0;
   // movePath.settings.movePathConfiguration.workspaceZones[1..10].zoneType := 0;
   // movePath.settings.movePathConfiguration.workspaceZones[1..10].coordinateSystem := 0;
   // movePath.settings.movePathConfiguration.workspaceZones[1..10].frame.x := 0.0;
   // movePath.settings.movePathConfiguration.workspaceZones[1..10].frame.y := 0.0;
   // movePath.settings.movePathConfiguration.workspaceZones[1..10].frame.z := 0.0;
   // movePath.settings.movePathConfiguration.workspaceZones[1..10].frame."a" := 0.0;
   // movePath.settings.movePathConfiguration.workspaceZones[1..10].frame."b" := 0.0;
   // movePath.settings.movePathConfiguration.workspaceZones[1..10].frame.c := 0.0;
   // movePath.settings.movePathConfiguration.workspaceZones[1..10].geometryType := 0;
   // movePath.settings.movePathConfiguration.workspaceZones[1].geometryParameter[1..3] := 0.0;
   // movePath.settings.movePathConfiguration.workspaceZones[2].geometryParameter[1..3] := 0.0;
   // movePath.settings.movePathConfiguration.workspaceZones[3].geometryParameter[1..3] := 0.0;
   // movePath.settings.movePathConfiguration.workspaceZones[4].geometryParameter[1..3] := 0.0;
   // movePath.settings.movePathConfiguration.workspaceZones[5].geometryParameter[1..3] := 0.0;
   // movePath.settings.movePathConfiguration.workspaceZones[6].geometryParameter[1..3] := 0.0;
   // movePath.settings.movePathConfiguration.workspaceZones[7].geometryParameter[1..3] := 0.0;
   // movePath.settings.movePathConfiguration.workspaceZones[8].geometryParameter[1..3] := 0.0;
   // movePath.settings.movePathConfiguration.workspaceZones[9].geometryParameter[1..3] := 0.0;
   // movePath.settings.movePathConfiguration.workspaceZones[10].geometryParameter[1..3] := 0.0;
   // movePath.settings.movePathConfiguration.kinematicsZones[1..10].coordinateSystem := 0;
   // movePath.settings.movePathConfiguration.kinematicsZones[1..10].frame.x := 0.0;
   // movePath.settings.movePathConfiguration.kinematicsZones[1..10].frame.y := 0.0;
   // movePath.settings.movePathConfiguration.kinematicsZones[1..10].frame.z := 0.0;
   // movePath.settings.movePathConfiguration.kinematicsZones[1..10].frame."a" := 0.0;
   // movePath.settings.movePathConfiguration.kinematicsZones[1..10].frame."b" := 0.0;
   // movePath.settings.movePathConfiguration.kinematicsZones[1..10].frame.c := 0.0;
   // movePath.settings.movePathConfiguration.kinematicsZones[1..10].geometryType := 0;
   // movePath.settings.movePathConfiguration.kinematicsZones[1].geometryParameter[1..3] := 0.0;
   // movePath.settings.movePathConfiguration.kinematicsZones[2].geometryParameter[1..3] := 0.0;
   // movePath.settings.movePathConfiguration.kinematicsZones[3].geometryParameter[1..3] := 0.0;
   // movePath.settings.movePathConfiguration.kinematicsZones[4].geometryParameter[1..3] := 0.0;
   // movePath.settings.movePathConfiguration.kinematicsZones[5].geometryParameter[1..3] := 0.0;
   // movePath.settings.movePathConfiguration.kinematicsZones[6].geometryParameter[1..3] := 0.0;
   // movePath.settings.movePathConfiguration.kinematicsZones[7].geometryParameter[1..3] := 0.0;
   // movePath.settings.movePathConfiguration.kinematicsZones[8].geometryParameter[1..3] := 0.0;
   // movePath.settings.movePathConfiguration.kinematicsZones[9].geometryParameter[1..3] := 0.0;
   // movePath.settings.movePathConfiguration.kinematicsZones[10].geometryParameter[1..3] := 0.0;
   // movePath.settings.movePathConfiguration.stopMode := 10;
   // movePath.settings.movePathConfiguration.interruptMode := 0;
   // movePath.transitionParameter[1] := -1.0;
END_TYPE
